{attribute addProperty BoxType "EJ5101-0000-0016"}
{attribute addProperty Id "StatusAT %I*Status_F0C09FF11621Counter_valueAT %I*UINT16217Latch_valueAT %I*UINT16218"}
{attribute addProperty CRC "1538259189"}
{attribute addProperty SizeInBites "48"}
{attribute addProperty SizeInBytes "6"}
TYPE ENC_Status_compact_5BAFF8F5 :
STRUCT
	{attribute addProperty Name "Status"}
	Status AT %I* : Status_F0C09FF1;
	{attribute addProperty Name "Counter_value"}
	Counter_value AT %I* : UINT;
	{attribute addProperty Name "Latch_value"}
	Latch_value AT %I* : UINT;
END_STRUCT
END_TYPE

(* stored: Version 1.2.0.0, ProductVersion 3.1.4024.9
   DUT ENC_Status_compact_5BAFF8F5: Id {0e374f2b-b1dc-4833-9701-ec9870eb6db6} *)
